TYPE ST_MoverFeedback :
STRUCT
	CallEnable			: MC_PlanarFeedback;
	CallDisable			: MC_PlanarFeedback;
	CallHalt			: MC_PlanarFeedback;
	CallJoinTrack		: MC_PlanarFeedback;
	CallLeaveTrack		: MC_PlanarFeedback;
	CallReset			: MC_PlanarFeedback;
	CallMoveX			: MC_PlanarFeedback;
	CallMoveY			: MC_PlanarFeedback;
	CallMoveZ			: MC_PlanarFeedback;
	CallMoveA			: MC_PlanarFeedback;
	CallMoveB			: MC_PlanarFeedback;
	CallMoveC			: MC_PlanarFeedback;
	CallMoveOnTrack		: MC_PlanarFeedback;
	CallEmergencyStop	: MC_PlanarFeedback;
	SeqJoinTrack		: MC_PlanarFeedback;
	
END_STRUCT
END_TYPE
//Feedback変数を構造体にして、Feedbackの名称を明示

(* stored: Version 1.1.0.1
   DUT ST_MoverFeedback: Id {38c98c8d-be9d-4a0b-8214-997bf5909abb} *)
